PROGRAM HMI
VAR
END_VAR

(*RESET SIMULATION*)
	IF GVL_HMI.bButtonResetSimilation THEN
		WaterTankFilling.fbTank.Reset();
		GVL_HMI.bButtonResetSimilation	:= FALSE;
	END_IF

(*TANK*)
	GVL_HMI.rTankMaxCapacity	:= WaterTankFilling.fbTank.rMaxCapacity;
	GVL_HMI.rTankCurrentLevel	:= WaterTankFilling.fbTank.rCurrentLevel;

(*LAMPS*)
	GVL_HMI.bLampPumpIsOn		:= WaterTankFilling.fbPump.bIsOn;
	GVL_HMI.bLampDrainValveIsOn	:= WaterTankFilling.fbDrainValve.bIsOn;
	
(*PUMP FLOW RATE*)
	GVL_HMI.rPumpActualFlowRate	:= WaterTankFilling.fbPump.rFlowRate;
	
	IF GVL_HMI.bButtonActualizePumpFlowRate THEN
		WaterTankFilling.fbPump.SetFlowRate(rRate := GVL_HMI.rPumpNewFlowRate);
		GVL_HMI.bButtonActualizePumpFlowRate	:= FALSE;
	END_IF

END_PROGRAM

(* stored: Version 1.1.0.1, ProductVersion 3.1.4024.12
   POU HMI: Id {5e4af75d-dd4b-41ee-a9bf-a1c1abbb42b8}, SpecialFunc None *)
